// TIA Portal V20 export
VAR_GLOBAL   // PLC tag table "Constantes de JDT01"
   Reintentos_JDT1 AT %MB8 : USInt;
END_VAR
VAR_GLOBAL CONSTANT   // user constants
   JDT1_FinalBucleMaquinas : UInt := 500;   // Ultima Maquina del JDT01
   JDT1_FinalBucleMesas : UInt := 500;   // Ultima Mesa del JDT01
   JDT1_IdentEmisor : DInt := 'PLC1';   // Identificador del Emisor MFS (JdT)
   JDT1_IdentReceptor : DInt := 'JDT1';   // Identificador del Receptor PLC
   JDT1_InicioBucleMaquinas : UInt := 1;   // Primera Maquina del JDT01
   JDT1_InicioBucleMesas : UInt := 1;   // Primera Mesa del JDT01
   JDT1_MaxBytes : UInt := 6000;   // Maximos numeros de Bytes para enviar o recibir por TCP (8192 Bytes)
   JDT1_NDB_AKEmi : UInt := 806;   // Numero de de la Emision AK
   JDT1_NDB_EmiMensaje : UInt := 803;   // Numero de DB de la Emisión del Mensaje hacia el MFS (JdT)
   JDT1_NDB_EventosEmi : UInt := 808;   // Numero de DB de la Lista de Eventos Generados
   JDT1_NDB_EventosRec : UInt := 807;   // Numero de DB de la Lista de Eventos Recibidos
   JDT1_NDB_RecMensaje : UInt := 802;   // Numero de DB de la Recepción del Mensaje del MFS (JdT)
   JDT1_NDB_UltimoEmi : UInt := 805;   // Numero de DB del Ultimo Mensaje Enviado
   JDT1_NDB_UltimoRec : UInt := 804;   // Numero de DB del Ultimo Mensaje Recibido
   JDT1_TMPEnvioKA : UInt := 60;   // Tiempo de Espera para el Envio del Keep-Alive - 1 Minuto
   JDT1_TMPEsperaAK : UInt := 10;   // Tiempo de Espera para recibir la Confirmacion del Mensaje Enviado - 10 Segundos
   JDT1_TMPEsperaKA : UInt := 120;   // Tiempo Maximo de Espera para recibir el Keep-Alive - 2 Minutos
END_VAR
